FUNCTION_BLOCK FB_Station01 EXTENDS FB_Station IMPLEMENTS IF_Station
VAR_INPUT
	//Ablauf
	//aReihenfolge:	ARRAY [1..Parameter.cAnzSchritte] OF AblaufStatus;  // über HMI befüllen
	aReihenfolge:	ARRAY [1..Parameter.cAnzSchritte] OF ST_Reihenfolge;
	fbAktor:		ARRAY [1..Parameter.cAnzAktoren] OF FB_Aktor[
											(bSensAPVorhanden:= FALSE, 
											bSensRPVorhanden:= FALSE, 
											tZeitRP:= T#3000MS, 
											tZeitAP:= T#3000MS, 
											nErrorIdAP:= 13, 
											nErrorIdRP:= 14, 
											sBezeichnung:= 'Aktor 1'),
											
											(bSensAPVorhanden:= FALSE, 
											bSensRPVorhanden:= FALSE, 
											tZeitRP:= T#3000MS, 
											tZeitAP:= T#3000MS, 
											nErrorIdAP:= 15, 
											nErrorIdRP:= 16, 
											sBezeichnung:= 'Aktor 2'),
											
											(bSensAPVorhanden:= FALSE, 
											bSensRPVorhanden:= FALSE, 
											tZeitRP:= T#3000MS, 
											tZeitAP:= T#3000MS, 
											nErrorIdAP:= 17, 
											nErrorIdRP:= 18, 
											sBezeichnung:= 'Aktor 3'),
											
											(bSensAPVorhanden:= FALSE, 
											bSensRPVorhanden:= FALSE, 
											tZeitRP:= T#3000MS, 
											tZeitAP:= T#3000MS, 
											nErrorIdAP:= 19, 
											nErrorIdRP:= 20, 
											sBezeichnung:= 'Aktor 4'),
											
											(bSensAPVorhanden:= FALSE, 
											bSensRPVorhanden:= FALSE, 
											tZeitRP:= T#3000MS, 
											tZeitAP:= T#3000MS, 
											nErrorIdAP:= 21, 
											nErrorIdRP:= 22, 
											sBezeichnung:= 'Aktor 5'),
											
											(bSensAPVorhanden:= FALSE, 
											bSensRPVorhanden:= FALSE, 
											tZeitRP:= T#3000MS, 
											tZeitAP:= T#3000MS, 
											nErrorIdAP:= 23, 
											nErrorIdRP:= 24, 
											sBezeichnung:= 'Aktor 6')
											];
	bSchrittbetriebAktiv:	BOOL;
	sNaechsterSchritt:		STRING;
END_VAR
VAR_OUTPUT
END_VAR
VAR


	
	//Inputs	
	bE_extGeraetBereit			AT%I*:	BOOL;

	bE_Sensor					AT %I* : ARRAY[1..8] OF BOOL;
	bA_extGeraetStart			AT%Q*:	BOOL;
	//Outputs

	//FBs	

	
	// Not-Halt testen täglich
	bNotHaltTestIO:			BOOL;
	fbNotHaltGedrueckt:		R_TRIG;
	bBtnResetWarnNothalt:	BOOL;
	bWarnungNothalt:		BOOL;
	bBtnResetAuftrZaehler:	BOOL;
	fbFlankeSchritt:		R_TRIG;
	bInit:					BOOL := TRUE;
	iSchritt:				INT := 1;								
	i: 						INT;
	x: 						INT;
	bSensorTeilAnwesend: 	BOOL;
	nStatusSchritt: 		INT;
	nZyklusZaehler:			INT;	
	
END_VAR

VAR_OUTPUT
	sStationsStatus:	STRING;
END_VAR

VAR PERSISTENT
	nMonatVorher:			WORD;
	nTagVorher:				WORD;
	nZaehlerNotHalt:		DINT;
END_VAR

fbFlankeSchritt(CLK := MAIN.bE_Taste_Schritt AND bSchrittbetriebAktiv);

//Array "aReihenfolge" mit dem Ablauf befüllen
IF			MAIN.HMI.bProgrammAngewaehlt 
		AND	reihenfolgeSchreiben() THEN
	MAIN.HMI.bProgrammAngewaehlt := FALSE;
END_IF

//********************************************************************************	
//Aktoren
fbAktor[1](fbSchrittbetrieb := fbSchrittbetrieb);
fbAktor[2](fbSchrittbetrieb := fbSchrittbetrieb);
fbAktor[3](fbSchrittbetrieb := fbSchrittbetrieb);
fbAktor[4](fbSchrittbetrieb := fbSchrittbetrieb);
fbAktor[5](fbSchrittbetrieb := fbSchrittbetrieb);
fbAktor[6](fbSchrittbetrieb := fbSchrittbetrieb); 



FOR x := 1 TO Parameter.cAnzAktoren DO
	IF			MAIN.HMI.ProgrammTemp.aAktorKonfig[x].nSensRuhePos > 0 THEN			
		fbAktor[x].bE_sensRP 	:= bE_Sensor[MAIN.HMI.ProgrammTemp.aAktorKonfig[x].nSensRuhePos];
		fbAktor[x].bSensRPVorhanden := TRUE;
	ELSE
		fbAktor[x].bSensRPVorhanden := FALSE;
	END_IF
	IF			MAIN.HMI.ProgrammTemp.aAktorKonfig[x].nSensArbeitsPos > 0 THEN			
		fbAktor[x].bE_sensAP 	:= bE_Sensor[MAIN.HMI.ProgrammTemp.aAktorKonfig[x].nSensArbeitsPos];
		fbAktor[x].bSensAPVorhanden := TRUE;
	ELSE
		fbAktor[x].bSensAPVorhanden := FALSE;
	END_IF	
	IF			MAIN.HMI.ProgrammTemp.aAktorKonfig[x].tFahrZeit = T#0MS THEN
		fbAktor[x].tZeitRP 		:= T#2000MS;
		fbAktor[x].tZeitAP 		:= T#2000MS;
	ELSE
		fbAktor[x].tZeitRP 		:= MAIN.HMI.ProgrammTemp.aAktorKonfig[x].tFahrZeit;
		fbAktor[x].tZeitAP 		:= MAIN.HMI.ProgrammTemp.aAktorKonfig[x].tFahrZeit;
	END_IF
	
	
END_FOR
	IF			bE_Sensor[MAIN.HMI.ProgrammTemp.nTeilAnw] THEN
		bSensorTeilAnwesend := TRUE;
	ELSE
		bSensorTeilAnwesend := FALSE;
	END_IF

FOR x := 1 TO Parameter.cAnzAktoren DO
	IF			NOT	stStationInfo.bInitBeendet THEN
		fbAktor[x].bSensRPVorhanden := FALSE;
		fbAktor[x].bSensAPVorhanden := FALSE;
	END_IF
END_FOR
		
//********************************************************************************	
//Sonstige FBs


//********************************************************************************
//Basisklasse ausführen
SUPER^(	stStationInfo := stStationInfo);


//********************************************************************************
//Stoerungen
stStationInfo.bStoerung := 			(fbAktor[1].bStoerung
							OR		fbAktor[2].bStoerung
							OR		fbAktor[3].bStoerung
							OR		fbAktor[4].bStoerung
							OR		fbAktor[5].bStoerung
							OR		fbAktor[6].bStoerung)
							AND		Main.bProduzieren
							AND NOT Main.bE_Handbetrieb;
							
sStationsStatus := stStationInfo.sStatus;

//********************************************************************************
//Warnung
stStationInfo.bWarnung := (			FALSE);

//Not-Halt-Test nach einem Tag zurücksetzen
IF		 	(nTagVorher <> MAIN.fbSystemZeit.TIMESTR.wDay 
	OR 	  	nMonatVorher <> MAIN.fbSystemZeit.TIMESTR.wMonth)
	AND		MAIN.fbSystemZeit.TIMESTR.wMonth > 0 THEN		//Damit der fbSystemzeit sicher ausgeführt wurde
	nTagVorher := MAIN.fbSystemZeit.TIMESTR.wDay;
	nMonatVorher := MAIN.fbSystemZeit.TIMESTR.wMonth;
	bNotHaltTestIO := FALSE;

END_IF

	// Not-Halt wurde betätigt
	IF		NOT	bNotHaltTestIO 
		AND	NOT	MAIN.bE_NotHalt THEN
		bNotHaltTestIO := TRUE;
	END_IF
	
	//Fehlermeldung
	IF		NOT bNotHaltTestIO
		AND	NOT	EventLogger.aAlarm[40].bRaised THEN
		EventLogger.aAlarm[40].Raise(0);
	ELSIF		bNotHaltTestIO
		AND		EventLogger.aAlarm[40].bRaised THEN
		EventLogger.aAlarm[40].Clear(0, TRUE);
	END_IF
	// Not-Halt Wartung
	fbNotHaltGedrueckt(CLK := NOT(MAIN.bE_NotHalt) AND MAIN.bInitBeendet);
	IF		fbNotHaltGedrueckt.Q THEN
		nZaehlerNotHalt := nZaehlerNotHalt + 1;
	END_IF
	IF		nZaehlerNotHalt >= Parameter.cMaxZyklNotHalt 
			AND	NOT	bWarnungNothalt THEN
		bWarnungNothalt := TRUE;
	END_IF
	
	IF		bBtnResetWarnNothalt 
		AND bWarnungNothalt THEN
			bBtnResetWarnNothalt := FALSE;
			bWarnungNothalt := FALSE;
			nZaehlerNotHalt := 0;
	END_IF

// Auftragszähler Reset
IF			bBtnResetAuftrZaehler THEN
	bBtnResetAuftrZaehler := FALSE;
	MAIN.stStueckzaehler.nAusschussAuftrag 	:= 0;
	MAIN.stStueckzaehler.nGutteileAuftrag 	:= 0;
END_IF

// Nächster Schritt auf HMI anzeigen im Schrittbetrieb

CASE aReihenfolge[iSchritt].eAblauf OF
	AblaufStatus.default:			sNaechsterSchritt := 'default';
	AblaufStatus.aktor01Vor:		sNaechsterSchritt := 'Aktor 1 vor';
	AblaufStatus.aktor01Zurueck:	sNaechsterSchritt := 'Aktor 1 zurück';
	AblaufStatus.aktor02Vor:		sNaechsterSchritt := 'Aktor 2 vor';
	AblaufStatus.aktor02Zurueck:	sNaechsterSchritt := 'Aktor 2 zurück';
	AblaufStatus.aktor03Vor:		sNaechsterSchritt := 'Aktor 3 vor';
	AblaufStatus.aktor03Zurueck:	sNaechsterSchritt := 'Aktor 3 zurück';
	AblaufStatus.aktor04Vor:		sNaechsterSchritt := 'Aktor 4 vor';
	AblaufStatus.aktor04Zurueck:	sNaechsterSchritt := 'Aktor 4 zurück';
	AblaufStatus.aktor05Vor:		sNaechsterSchritt := 'Aktor 5 vor';
	AblaufStatus.aktor05Zurueck:	sNaechsterSchritt := 'Aktor 5 zurück';
	AblaufStatus.aktor06Vor:		sNaechsterSchritt := 'Aktor 6 vor';
	AblaufStatus.aktor06Zurueck:	sNaechsterSchritt := 'Aktor 6 zurück';
	AblaufStatus.teilAnwesend:		sNaechsterSchritt := 'teilAnwesend';
	AblaufStatus.bereit:			sNaechsterSchritt := 'bereit';
	AblaufStatus.error:				sNaechsterSchritt := 'error';
	AblaufStatus.extGeraetBereit:	sNaechsterSchritt := 'extGeraetBereit';
	AblaufStatus.extGeraetFertig:	sNaechsterSchritt := 'extGeraetFertig';
	AblaufStatus.extGeraetStart:	sNaechsterSchritt := 'extGeraetStart';
	AblaufStatus.fertig:			sNaechsterSchritt := 'fertig';
	AblaufStatus.warten:			sNaechsterSchritt := 'warten';
END_CASE



//************************************************************************
//Muss alles nach dem Ablauf sein, damit das Main die Aktuellen Werte hat.
//************************************************************************

//Zyklus Fertig	
stStationInfo.bZyklusFertig :=		NOT bTeilBearbeiten;
bInit := FALSE;

METHOD ablaufSchreiben : AblaufStatus
VAR_INPUT
END_VAR

VAR
	eAblaufStatus: AblaufStatus;
	i:		INT := 1;
END_VAR

// Ablauf aus ARRAY Reihenfolge in AblaufStatus schreiben
// Wenn beim Aktor Pendelbetrieb aktiviert ist, muss der Ablaufstatus jedes Mal wechseln zwischen den Zyklen, z.B. aktor01Vor <> aktor02Zurueck
// Dies wird z.B bei einer Verdrillvorrichtung für den RST benötigt
// MAIN.HMI.ProgrammTemp.aAktorKonfig[1]


IF			nZyklusZaehler = 0 THEN
	// Ablauf für Aktoren korrigieren gemäss ihrem aktuellen Zustand
		IF			fbAktor[1].inAP()
			AND		aReihenfolge[iSchritt].eAblauf = AblaufStatus.aktor01Vor THEN
				eAblaufStatus := AblaufStatus.aktor01Zurueck;
//		ELSIF 		fbAktor[1].inRP()
//			AND		aReihenfolge[iSchritt].eAblauf = AblaufStatus.aktor01Zurueck THEN
//				eAblaufStatus := AblaufStatus.aktor01Vor;
				
		ELSIF 		fbAktor[2].inAP()
			AND		aReihenfolge[iSchritt].eAblauf = AblaufStatus.aktor02Vor THEN
				eAblaufStatus := AblaufStatus.aktor02Zurueck;
//		ELSIF 		fbAktor[2].inRP()
//			AND		aReihenfolge[iSchritt].eAblauf = AblaufStatus.aktor02Zurueck THEN
//				eAblaufStatus := AblaufStatus.aktor02Vor;
		
		ELSIF 		fbAktor[3].inAP()
			AND		aReihenfolge[iSchritt].eAblauf = AblaufStatus.aktor03Vor THEN
				eAblaufStatus := AblaufStatus.aktor03Zurueck;
				
		ELSIF 		fbAktor[4].inAP()
			AND		aReihenfolge[iSchritt].eAblauf = AblaufStatus.aktor04Vor THEN
				eAblaufStatus := AblaufStatus.aktor04Zurueck;
				
		ELSIF 		fbAktor[5].inAP()
			AND		aReihenfolge[iSchritt].eAblauf = AblaufStatus.aktor05Vor THEN
				eAblaufStatus := AblaufStatus.aktor05Zurueck;
				
		ELSIF 		fbAktor[6].inAP()
			AND		aReihenfolge[iSchritt].eAblauf = AblaufStatus.aktor06Vor THEN
				eAblaufStatus := AblaufStatus.aktor06Zurueck;
				
		ELSE
			eAblaufStatus := aReihenfolge[iSchritt].eAblauf;
		END_IF


	//eAblaufStatus := aReihenfolge[iSchritt].eAblauf;
	aReihenfolge[iSchritt].eLetzterStatus := eAblaufStatus;
	
ELSE
	CASE aReihenfolge[iSchritt].eLetzterStatus OF
		
		//****************************************************************************************	
		//****************************************************************************************
		AblaufStatus.aktor01Vor:
			IF			MAIN.HMI.ProgrammTemp.aAktorKonfig[1].bReversierBetrieb THEN
				eAblaufStatus := AblaufStatus.aktor01Zurueck;
			ELSE
				eAblaufStatus := AblaufStatus.aktor01Vor;
			END_IF
			aReihenfolge[iSchritt].eLetzterStatus := eAblaufStatus;
			
		//****************************************************************************************	
		AblaufStatus.aktor01Zurueck:
			IF			MAIN.HMI.ProgrammTemp.aAktorKonfig[1].bReversierBetrieb THEN
				eAblaufStatus := AblaufStatus.aktor01Vor;
			ELSE
				eAblaufStatus := AblaufStatus.aktor01Zurueck;
			END_IF
			aReihenfolge[iSchritt].eLetzterStatus := eAblaufStatus;
			
		//****************************************************************************************	
		//****************************************************************************************
		AblaufStatus.aktor02Vor:
			IF			MAIN.HMI.ProgrammTemp.aAktorKonfig[2].bReversierBetrieb THEN
				eAblaufStatus := AblaufStatus.aktor02Zurueck;
			ELSE
				eAblaufStatus := AblaufStatus.aktor02Vor;
			END_IF
			aReihenfolge[iSchritt].eLetzterStatus := eAblaufStatus;
			
		//****************************************************************************************	
		AblaufStatus.aktor02Zurueck:
			IF			MAIN.HMI.ProgrammTemp.aAktorKonfig[2].bReversierBetrieb THEN
				eAblaufStatus := AblaufStatus.aktor02Vor;
			ELSE
				eAblaufStatus := AblaufStatus.aktor02Zurueck;
			END_IF	
			aReihenfolge[iSchritt].eLetzterStatus := eAblaufStatus;
			
		//****************************************************************************************	
		//****************************************************************************************
		AblaufStatus.aktor03Vor:
			IF			MAIN.HMI.ProgrammTemp.aAktorKonfig[3].bReversierBetrieb THEN
				eAblaufStatus := AblaufStatus.aktor03Zurueck;
			ELSE
				eAblaufStatus := AblaufStatus.aktor03Vor;
			END_IF
			aReihenfolge[iSchritt].eLetzterStatus := eAblaufStatus;
			
		//****************************************************************************************	
		AblaufStatus.aktor03Zurueck:
			IF			MAIN.HMI.ProgrammTemp.aAktorKonfig[3].bReversierBetrieb THEN
				eAblaufStatus := AblaufStatus.aktor03Vor;
			ELSE
				eAblaufStatus := AblaufStatus.aktor03Zurueck;
			END_IF
			aReihenfolge[iSchritt].eLetzterStatus := eAblaufStatus;
			
		//****************************************************************************************	
		//****************************************************************************************
		AblaufStatus.aktor04Vor:
			IF			MAIN.HMI.ProgrammTemp.aAktorKonfig[4].bReversierBetrieb THEN
				eAblaufStatus := AblaufStatus.aktor04Zurueck;
			ELSE
				eAblaufStatus := AblaufStatus.aktor04Vor;
			END_IF
			aReihenfolge[iSchritt].eLetzterStatus := eAblaufStatus;
			
		//****************************************************************************************	
		AblaufStatus.aktor04Zurueck:
			IF			MAIN.HMI.ProgrammTemp.aAktorKonfig[4].bReversierBetrieb THEN
				eAblaufStatus := AblaufStatus.aktor04Vor;
			ELSE
				eAblaufStatus := AblaufStatus.aktor04Zurueck;
			END_IF
			aReihenfolge[iSchritt].eLetzterStatus := eAblaufStatus;
			
		//****************************************************************************************	
		//****************************************************************************************
		AblaufStatus.aktor05Vor:
			IF			MAIN.HMI.ProgrammTemp.aAktorKonfig[5].bReversierBetrieb THEN
				eAblaufStatus := AblaufStatus.aktor05Zurueck;
			ELSE
				eAblaufStatus := AblaufStatus.aktor05Vor;
			END_IF
			aReihenfolge[iSchritt].eLetzterStatus := eAblaufStatus;
			
		//****************************************************************************************	
		AblaufStatus.aktor05Zurueck:
			IF			MAIN.HMI.ProgrammTemp.aAktorKonfig[5].bReversierBetrieb THEN
				eAblaufStatus := AblaufStatus.aktor05Vor;
			ELSE
				eAblaufStatus := AblaufStatus.aktor05Zurueck;
			END_IF
			aReihenfolge[iSchritt].eLetzterStatus := eAblaufStatus;
			
		//****************************************************************************************	
		//****************************************************************************************
		AblaufStatus.aktor06Vor:
			IF			MAIN.HMI.ProgrammTemp.aAktorKonfig[6].bReversierBetrieb THEN
				eAblaufStatus := AblaufStatus.aktor06Zurueck;
			ELSE
				eAblaufStatus := AblaufStatus.aktor06Vor;
			END_IF
			aReihenfolge[iSchritt].eLetzterStatus := eAblaufStatus;
			
		//****************************************************************************************	
		AblaufStatus.aktor06Zurueck:
			IF			MAIN.HMI.ProgrammTemp.aAktorKonfig[6].bReversierBetrieb THEN
				eAblaufStatus := AblaufStatus.aktor06Vor;
			ELSE
				eAblaufStatus := AblaufStatus.aktor06Zurueck;
			END_IF
			aReihenfolge[iSchritt].eLetzterStatus := eAblaufStatus;	
	ELSE
			eAblaufStatus := aReihenfolge[iSchritt].eAblauf;
			
	END_CASE	
END_IF


ablaufSchreiben := eAblaufStatus;
END_METHOD

METHOD init : BOOL
CASE eInitStatus OF
	//***********************************************************************************************
	InitStatus.bereit:
			
		IF 		NOT stStationInfo.bInitBeendet THEN
			EventLogger.aMessage[10].ipArguments.Clear().AddString('Aktoren');
			EventLogger.aMessage[10].Send(0);
			bTeilBearbeiten := FALSE;									// Hier richtig?
			eInitStatus := InitStatus.aktor1;
		END_IF
		
	//***********************************************************************************************
	InitStatus.aktor1:
		
		IF		fbAktor[1].ruhePos() THEN
			eInitStatus := InitStatus.aktor2;
		END_IF

	//***********************************************************************************************
	InitStatus.aktor2:
	
		IF		fbAktor[2].ruhePos() THEN
			eInitStatus := InitStatus.aktor3;
		END_IF

	//***********************************************************************************************
	InitStatus.aktor3:
	
		IF		fbAktor[3].ruhePos() THEN
			eInitStatus := InitStatus.aktor4;
		END_IF

	//***********************************************************************************************
	InitStatus.aktor4:
	
		IF		fbAktor[4].ruhePos() THEN
			eInitStatus := InitStatus.aktor5;
		END_IF

	//***********************************************************************************************
	InitStatus.aktor5:
	
		IF		fbAktor[5].ruhePos() THEN
			eInitStatus := InitStatus.aktor6;
		END_IF

	//***********************************************************************************************
	InitStatus.aktor6:	
	
		IF		fbAktor[6].ruhePos() THEN
			eInitStatus := InitStatus.fertig;
		END_IF
	
	//***********************************************************************************************
	InitStatus.fertig:
		
		EventLogger.aMessage[11].Send(0);
		
		stStationInfo.bInitBeendet := TRUE;
		MAIN.bProduzieren := FALSE;
		eInitStatus := InitStatus.bereit;
	
END_CASE

init := stStationInfo.bInitBeendet;
END_METHOD

METHOD reihenfolgeSchreiben : bool
VAR_INPUT
END_VAR
nZyklusZaehler := 0;

FOR i := 1 TO Parameter.cAnzSchritte DO	 	
	
	aReihenfolge[i].eAblauf := MAIN.HMI.ProgrammTemp.aAktorBew[i].eAblaufStatus;

	// Den Aktoren die Zeiten zuweisen aus dem Programm
	IF			aReihenfolge[i].eAblauf = Ablaufstatus.aktor01Vor
		OR		aReihenfolge[i].eAblauf = Ablaufstatus.aktor01Zurueck THEN
			aReihenfolge[i].tFahrzeit := MAIN.HMI.ProgrammTemp.aAktorKonfig[1].tFahrZeit;
			aReihenfolge[i].tHalteZeit := MAIN.HMI.ProgrammTemp.aAktorKonfig[1].tHalteZeit;
			
	ELSIF		aReihenfolge[i].eAblauf = Ablaufstatus.aktor02Vor
		OR		aReihenfolge[i].eAblauf = Ablaufstatus.aktor02Zurueck THEN
			aReihenfolge[i].tFahrzeit := MAIN.HMI.ProgrammTemp.aAktorKonfig[2].tFahrZeit;
			aReihenfolge[i].tHalteZeit := MAIN.HMI.ProgrammTemp.aAktorKonfig[2].tHalteZeit;
	
	ELSIF		aReihenfolge[i].eAblauf = Ablaufstatus.aktor03Vor
		OR		aReihenfolge[i].eAblauf = Ablaufstatus.aktor03Zurueck THEN
			aReihenfolge[i].tFahrzeit := MAIN.HMI.ProgrammTemp.aAktorKonfig[3].tFahrZeit;
			aReihenfolge[i].tHalteZeit := MAIN.HMI.ProgrammTemp.aAktorKonfig[3].tHalteZeit;
			
	ELSIF		aReihenfolge[i].eAblauf = Ablaufstatus.aktor04Vor
		OR		aReihenfolge[i].eAblauf = Ablaufstatus.aktor04Zurueck THEN
			aReihenfolge[i].tFahrzeit := MAIN.HMI.ProgrammTemp.aAktorKonfig[4].tFahrZeit;
			aReihenfolge[i].tHalteZeit := MAIN.HMI.ProgrammTemp.aAktorKonfig[4].tHalteZeit;
			
	ELSIF		aReihenfolge[i].eAblauf = Ablaufstatus.aktor05Vor
		OR		aReihenfolge[i].eAblauf = Ablaufstatus.aktor05Zurueck THEN
			aReihenfolge[i].tFahrzeit := MAIN.HMI.ProgrammTemp.aAktorKonfig[5].tFahrZeit;
			aReihenfolge[i].tHalteZeit := MAIN.HMI.ProgrammTemp.aAktorKonfig[5].tHalteZeit;
			
	ELSIF		aReihenfolge[i].eAblauf = Ablaufstatus.aktor06Vor
		OR		aReihenfolge[i].eAblauf = Ablaufstatus.aktor06Zurueck THEN
			aReihenfolge[i].tFahrzeit := MAIN.HMI.ProgrammTemp.aAktorKonfig[6].tFahrZeit;
			aReihenfolge[i].tHalteZeit := MAIN.HMI.ProgrammTemp.aAktorKonfig[6].tHalteZeit;
	END_IF
END_FOR	

reihenfolgeSchreiben := TRUE;
END_METHOD

METHOD reset : BOOL
CASE eResetStatus OF
	
	//***********************************************************************************************
	ResetStatus.bereit:
		
		eResetStatus := ResetStatus.ablaufAbbrechen;
		iSchritt := 1;
		
	//***********************************************************************************************
	ResetStatus.ablaufAbbrechen:
		
		eAblaufStatus 		:= AblaufStatus.bereit;
		fbSchrittbetrieb.reset();
		eResetStatus 		:= ResetStatus.aktoren;
	

		
	//***********************************************************************************************
	ResetStatus.aktoren:	
		FOR i:= 1 TO Parameter.cAnzAktoren DO
			fbAktor[i].bHandOverride := NOT MAIN.bE_SafetyProgStop;
			IF			fbAktor[i].ruhePos() THEN
				eResetStatus 		:= ResetStatus.fertig;
				fbAktor[i].bHandOverride := FALSE;
			END_IF
		END_FOR
	
	//***********************************************************************************************
	ResetStatus.fertig:
		
		eInitStatus := InitStatus.bereit;
		
		IF 			stStationInfo.bInitBeendet THEN		//Wenn schon initialisiert wurde, wird ein reinit durchgeführt
			stStationInfo.bInit := TRUE;				//War die Station schon am init, wurde bInit nie false und das init startet erneut
			stStationInfo.bInitBeendet := FALSE;
		END_IF
		
		reset := TRUE;
END_CASE
END_METHOD

METHOD teilBearbeiten : BOOL
VAR_INST
	//fbMessage:	FB_Message;
	fbTon:		TON;
	fbTonHalten:	TON;
	tTime:		TIME;
END_VAR
CASE eAblaufStatus OF
	
	AblaufStatus.bereit:
		IF			fbFlankeSchritt.Q 
			OR NOT	bSchrittbetriebAktiv THEN
			eAblaufStatus := AblaufStatus.schritt;
		END_IF
		
//****************************************************************************************
	AblaufStatus.schritt:		
		IF			aReihenfolge[iSchritt].eAblauf <> 	AblaufStatus.default  THEN
			eAblaufStatus := ablaufSchreiben();
			//eAblaufStatus := aReihenfolge[iSchritt].eAblauf;						// wird über Methode "ablaufSchreiben" erledigt
			fbTon(IN := FALSE, PT := aReihenfolge[iSchritt].tFahrzeit);		
			fbTonHalten(IN := FALSE, PT := aReihenfolge[iSchritt].tHaltezeit);	
		ELSE
			eAblaufStatus := AblaufStatus.fertig;
			nZyklusZaehler := nZyklusZaehler + 1;
			iSchritt := 1;
		END_IF
		
	//****************************************************************************************
	AblaufStatus.aktor01Vor:
	
		IF			fbAktor[1].arbeitsPos() THEN
			eAblaufStatus := AblaufStatus.naechsterSchritt;
		END_IF
	
	//****************************************************************************************
	AblaufStatus.aktor01Zurueck:
	
		IF			fbAktor[1].ruhePos() THEN
			eAblaufStatus := AblaufStatus.naechsterSchritt;
		END_IF
	
	//****************************************************************************************
	AblaufStatus.aktor02Vor:
	
		IF			fbAktor[2].arbeitsPos() THEN
			eAblaufStatus := AblaufStatus.naechsterSchritt;
		END_IF
	
	//****************************************************************************************
	AblaufStatus.aktor02Zurueck:
	
		IF			fbAktor[2].ruhePos() THEN
			eAblaufStatus := AblaufStatus.naechsterSchritt;
		END_IF

	//****************************************************************************************
	AblaufStatus.aktor03Vor:
	
		IF			fbAktor[3].arbeitsPos() THEN
			eAblaufStatus := AblaufStatus.naechsterSchritt;
		END_IF
	
	//****************************************************************************************
	AblaufStatus.aktor03Zurueck:
	
		IF			fbAktor[3].ruhePos() THEN
			eAblaufStatus := AblaufStatus.naechsterSchritt;
		END_IF

	//****************************************************************************************
	AblaufStatus.aktor04Vor:
	
		IF			fbAktor[4].arbeitsPos() THEN
			eAblaufStatus := AblaufStatus.naechsterSchritt;
		END_IF
	
	//****************************************************************************************
	AblaufStatus.aktor04Zurueck:
	
		IF			fbAktor[4].ruhePos() THEN
			eAblaufStatus := AblaufStatus.naechsterSchritt;
		END_IF

	//****************************************************************************************
	AblaufStatus.aktor05Vor:
	
		IF			fbAktor[5].arbeitsPos() THEN
			eAblaufStatus := AblaufStatus.naechsterSchritt;
		END_IF
	
	//****************************************************************************************
	AblaufStatus.aktor05Zurueck:	
	
		IF			fbAktor[5].ruhePos() THEN
			eAblaufStatus := AblaufStatus.naechsterSchritt;
		END_IF

	//****************************************************************************************
	AblaufStatus.aktor06Vor:
	
		IF			fbAktor[6].arbeitsPos() THEN
			eAblaufStatus := AblaufStatus.naechsterSchritt;
		END_IF
	
	//****************************************************************************************
	AblaufStatus.aktor06Zurueck:	
	
		IF			fbAktor[6].ruhePos() THEN
			eAblaufStatus := AblaufStatus.naechsterSchritt;
		END_IF
		
	//***********************************************************************************************
	AblaufStatus.warten:	
		
		fbTon(IN := TRUE);
		IF			fbton.Q THEN
			eAblaufStatus := AblaufStatus.naechsterSchritt;
		END_IF
		
	//***********************************************************************************************
	AblaufStatus.error:

			eAblaufStatus := AblaufStatus.naechsterSchritt;

	//***********************************************************************************************
	AblaufStatus.extGeraetBereit:

		IF		bE_extGeraetBereit	THEN
			eAblaufStatus := AblaufStatus.naechsterSchritt;
		END_IF
		
	//***********************************************************************************************
	AblaufStatus.extGeraetStart:
		
		bA_extGeraetStart := TRUE;
		IF		NOT	bE_extGeraetBereit	THEN
			eAblaufStatus := AblaufStatus.extGeraetFertig;		
		END_IF	
		
	//***********************************************************************************************
	AblaufStatus.extGeraetFertig:
		IF		bE_extGeraetBereit	THEN
			eAblaufStatus := AblaufStatus.naechsterSchritt;
			bA_extGeraetStart := FALSE;
		END_IF
			
	//***********************************************************************************************		
	AblaufStatus.teilAnwesend:
		
		IF			bSensorTeilAnwesend THEN
			eAblaufStatus := AblaufStatus.naechsterSchritt;	
		END_IF
	
	//***********************************************************************************************
	AblaufStatus.naechsterSchritt:
	
		fbTonHalten(IN := TRUE);
		IF			fbTonHalten.Q 
			AND NOT	MAIN.bE_Taste_Schritt THEN
			iSchritt := iSchritt + 1;
			eAblaufStatus := AblaufStatus.bereit;
		END_IF
		
	//***********************************************************************************************
	AblaufStatus.fertig:		
	
			eAblaufStatus := AblaufStatus.bereit;
			teilbearbeiten := TRUE;
			MAIN.bProduzieren := FALSE;
			MAIN.zaehlerGut();
		
END_CASE
END_METHOD

END_FUNCTION_BLOCK

(* stored: Version 1.1.0.1, ProductVersion 3.1.4024.12
   POU FB_Station01: Id {7b42e531-f381-47bd-ac94-8ae1c13c3c43}, SpecialFunc None
   Method ablaufSchreiben: Id {a2c5d6ea-3643-454c-9da6-50669ac3209b}
   Method init: Id {319694de-c8f1-48d6-91e1-37a51046f423}
   Method reihenfolgeSchreiben: Id {e1e7a774-99fb-4024-b8ea-7ad7dc842121}
   Method reset: Id {25cad2b3-7140-40c3-b6e8-4829d71ebb68}
   Method teilBearbeiten: Id {72a7a9ec-952e-47e9-b71f-088564088e8a} *)
